// TIA Portal V20 export
FUNCTION_BLOCK "SafetyCom"   // FB45, FBD
{ S7_Optimized_Access := 'TRUE' }
// stored: AutoNumber false, MemoryReserve 100, SetENOAutomatically false
   VAR DB_SPECIFIC
      Var { ExternalAccessible := 'False'; ExternalVisible := 'False'; ExternalWritable := 'False'} : "TypeVar";
   END_VAR
BEGIN

REGION Network 1 (SCL): reset important data if communication is not working
   IF "G".errComPc THEN
       "ComRd".Data.safety.AreaAdjustmentOn := FALSE;
       "ComRd".Data.safety.AreaLaserOn := FALSE;
       "ComRd".Data.safety.AreaXrayOn  := FALSE;
       "ComRd".Data.safety.ResetSafetyDevice := FALSE;
   END_IF;
END_REGION

REGION Network 2 (SCL): safety program - copy data
   "SiCom".Ack := "G".ack;
   "SiCom".Blinker := "blinker";
   "SiCom".Flash := "flash";
   "SiCom".LampTest.SettingMode:= "ComRd".Data.TestOutput.Active AND "ComRd".Data.TestOutput."Q900.1";
   "SiCom".LampTest.LaserOn := "ComRd".Data.TestOutput.Active AND "ComRd".Data.TestOutput."Q908.0";
   "SiCom".LampTest.XrayOn := "ComRd".Data.TestOutput.Active AND "ComRd".Data.TestOutput."Q908.1";
   "SiCom".SafetyTest := false;

   "SiCom".AreaAdjustmentOn := "ComRd".Data.safety.AreaAdjustmentOn OR TRUE;
   "SiCom".AreaLaserOn := "ComRd".Data.safety.AreaLaserOn;
   "SiCom".AreaXrayOn := "ComRd".Data.safety.AreaXrayOn;

   "SiCom".ResetSafetyDevice := "ComRd".Data.safety.ResetSafetyDevice OR "G".ack;
END_REGION
END_FUNCTION_BLOCK
